# EPICS substitutions: zfmagfldSup/zfmagfld_sensor_matrix.substitutions
file zfmagfld_sensor_matrix.template {
  pattern
    {P, ROW, COLUMN}

    {"\$(P)", "1", "1",}
    {"\$(P)", "1", "2",}
    {"\$(P)", "1", "3",}

    {"\$(P)", "2", "1",}
    {"\$(P)", "2", "2",}
    {"\$(P)", "2", "3",}

    {"\$(P)", "3", "1",}
    {"\$(P)", "3", "2",}
    {"\$(P)", "3", "3",}
}
